# EPICS SNL sequencer program: siteApps/SCL3Cooldown-sim-2-O/cooldownApp/src/CDFanoutTest.stt
program CDFanoutTest
option +r;

%% #include <math.h>

int proc;
assign proc "SCL3-CoolDown:FwdLnk.PROC";

ss steadystate
{
	state init
	{
		when(TRUE)
		{
			//initialization
			proc = 1;
			pvPut(proc, SYNC);
		} state processing
	}

	state processing
	{
		when(delay(5.0))
		{
			proc = 1;
			pvPut(proc, SYNC);
		}state processing
	}

}
